// TIA Portal V17 export
// export: Created 2025-03-07T09:19:46.8362116Z, ExportSetting WithDefaults, DisplayName Totally Integrated Automation Portal, DisplayVersion V17 Update 8, DisplayName TIA Portal Openness, DisplayVersion V17 Update 8, DisplayName TIA Portal Version Control Interface, DisplayVersion V17, DisplayName SINAMICS Startdrive Advanced, DisplayVersion V17 SP2, DisplayName SINAMICS Startdrive G110M, G120, G120C, G120D, G120P, G115D, DisplayVersion V17 SP2, DisplayName SINAMICS Startdrive G130, G150, S120, S150, SINAMICS MV, S210, DisplayVersion V17 SP2, DisplayName STEP 7 Professional, DisplayVersion V17 Update 8, DisplayName SINUMERIK ONE STEP 7 Toolbox, DisplayVersion V17 Update 12, DisplayName SINUMERIK 840D sl STEP 7 Toolbox, DisplayVersion V17 Update 12, DisplayName STEP 7 Safety, DisplayVersion V17 Update 6, DisplayName WinCC Advanced, DisplayVersion V17 Update 8
TYPE "MODES"
// stored: IsFailsafeCompliant false
   STRUCT
      GENERAL_CONDITIONS : Bool;   // CHANGE GENERAL CONDITIONS / GENERAL CONDITIONS
      INITIAL_CONDITIONS : Bool;   // CHANGE INITIAL CONDITIONS / INITIAL CONDITIONS
      ENABLE_REQUEST : Bool;   // ENABLE REQUEST
      DISABLE_REQUEST : Bool;   // DISABLE REQUEST
      TOGGLE_COMMAND_P : Bool;   // TOGGLE COMAND PULSE / TOGGLE COMMAND PULSE
      TOGGLE_COMMAND : Bool;   // TOGGLE COMMAND AUXILIARY / TOGGLE COMMAND
      GENERAL_CONDITIONS_HELP : Bool;   // GENERAL CONDITIONS HELP
      INITIAL_CONDITIONS_HELP : Bool;   // INITIAL CONDITIONS HELP
      MODE_SELECTED : Bool;   // MODE SELECTED
      WARNING_GONE : Bool;   // WARNING GONE
   END_STRUCT;
END_TYPE
